# EPICS autosave request: iocBoot/iocTomoScanFPGA_2BMB/auto_settings.req
file "tomoScan_settings.req", P=$(P), R=$(R)
file "tomoScan_PSO_settings.req", P=$(P), R=$(R)
file "tomoScan_2BM_settings.req", P=$(P), R=$(R)
file "tomoScan_FPGA_settings.req", P=$(P), R=$(R)
